TYPE ST_InfluxAlarmsRetrieve :
STRUCT
    {attribute 'TagName' := 'time'}
	MesTime			: LINT;
    {attribute 'TagName' := 'Message'}
	Message		 	: T_MaxString;	// Alarm Message 
    {attribute 'FieldName' := 'ID'}	
	ID				: ULINT;
    {attribute 'FieldName' := 'Value'}	
	Value 			: BOOL;
    {attribute 'FieldName' := 'Ack'}	
	Ack				: BOOL;	
END_STRUCT
END_TYPE

(* stored: Version 1.1.0.1, ProductVersion 3.1.4024.6
   DUT ST_InfluxAlarmsRetrieve: Id {2cd5e29d-7396-4d04-8653-0e50f0b65027} *)
